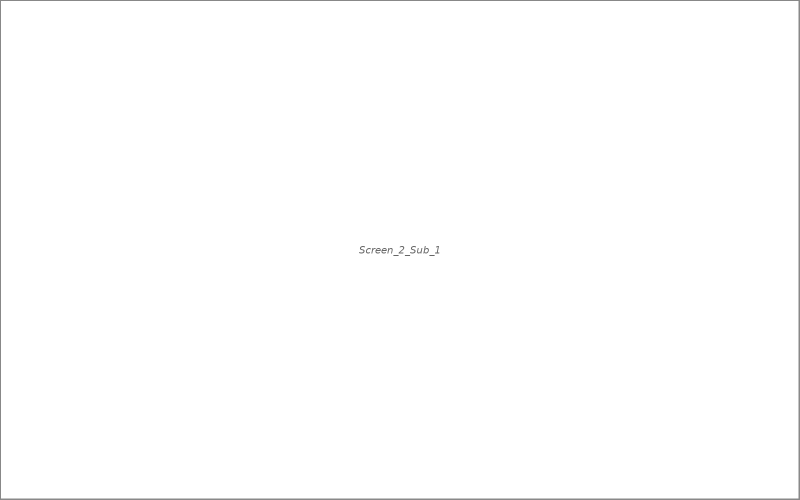
VISUALIZATION Screen_2  // 800x500
    TabControl (0,0 800x500), frame switch variable: GVL.HMI_Heading[2]
        shows Screen_2_Sub_1()
        shows Screen_2_Sub_2()
        shows Screen_2_Sub_6()
        shows Screen_2_Sub_3()
        shows Screen_2_Sub_4()
        shows Screen_2_Sub_7()
        shows Screen_2_Sub_5()
        [0]: TabTitle=Motor Peristaltik
        [1]: TabTitle=Motor DAC 1
        [2]: TabTitle=Motor DAC 2
        [3]: TabTitle=Motor Pump 1
        [4]: TabTitle=Motor Pump 2
        [5]: TabTitle=Motor Pump 3
        [6]: TabTitle=Motor Stepper
END_VISUALIZATION

(* stored: Version 1.1.0.1, ProductVersion 3.1.4024.12
   Visu Screen_2: Id {53c664e4-ed94-41c0-9198-b99221469e4b} *)
